Yaskawa INFORM job: TCP_LONG_SPIKE2.JBI

/JOB
//NAME TCP_LONG_SPIKE2
///FOLDERNAME INNE
//POS
///NPOS 15,15,0,0,0,0
///TOOL 0
///POSTYPE PULSE
///PULSE
C00000=-1196,10767,86976,6877,108771,41684
C00001=55051,-14614,53026,5978,107263,52173
C00002=127084,-16099,51982,6316,107113,52295
C00003=164428,-21371,45377,7399,109099,42690
C00004=223137,-21242,45410,8249,109054,43021
C00005=-230450,-1959,70810,8514,108912,45297
C00006=-149283,6312,81136,8104,106754,51735
C00007=-120085,293,72434,8477,110154,40524
C00008=-43968,-13280,53822,-6576,113295,-26885
C00009=-64332,-52250,7607,-6892,102968,-37506
C00010=-174949,-38434,23505,-6038,105852,-42530
C00011=-224736,-80728,-16448,-1859,96147,-10777
C00012=-24375,-110749,-34739,6827,71520,34674
C00013=39798,-71080,-9373,4554,90372,59950
C00014=-1529,-47599,12704,6701,104210,40081
BC00000=234605,127399,695029
BC00001=234605,127399,695029
BC00002=234605,127399,695029
BC00003=234605,127399,695029
BC00004=234605,127399,695029
BC00005=234605,127399,695029
BC00006=234605,127399,695029
BC00007=234605,127399,695029
BC00008=234605,127399,695029
BC00009=234605,127399,695029
BC00010=234605,127399,695029
BC00011=234605,127399,695029
BC00012=234605,127399,695029
BC00013=234605,127399,695029
BC00014=234605,127399,695029
//INST
///DATE 2023/10/04 15:16
///ATTR SC,RW
///GROUP1 RB1,BS1
NOP
MOVJ C00000 BC00000 VJ=0.78
MOVJ C00001 BC00001 VJ=0.78
MOVJ C00002 BC00002 VJ=0.78
MOVJ C00003 BC00003 VJ=0.78
MOVJ C00004 BC00004 VJ=0.78
MOVJ C00005 BC00005 VJ=0.78
MOVJ C00006 BC00006 VJ=0.78
MOVJ C00007 BC00007 VJ=0.78
MOVJ C00008 BC00008 VJ=0.78
MOVJ C00009 BC00009 VJ=0.78
MOVJ C00010 BC00010 VJ=0.78
MOVJ C00011 BC00011 VJ=0.78
MOVJ C00012 BC00012 VJ=0.78
MOVJ C00013 BC00013 VJ=0.78
MOVJ C00014 BC00014 VJ=0.78
END
